(* Logix 5000 project; controller fun_probably 1769-L16ER-BB1B rev 34.12; software revision 34.01 *)

TASK MainTask (continuous, watchdog 500 ms) : MainProgram

MODULES
   Local : 1769-L16ER-BB1B (PointIO 0, rev 34.12)
      Discrete_IO : Embedded (PointIO 1, rev 34.11, Output RPI 20 ms)
END_MODULES

VAR_GLOBAL   (* controller tags *)
   ball_move : BOOL;
   ballSpeed : DINT;
   ballSpeedX : DINT := 4;
   ballSpeedY : DINT := 3;
   ballXpos : COUNTER := (ACC := 225);
   ballYpos : COUNTER := (ACC := 100);
   difficulty : TIMER := (PRE := 5000, ACC := 4915, EN := 1, TT := 1);
   direction : DINT;
   directionX : DINT := 1;
   directionY : DINT := 1;
   dX : DINT := 6;
   dY : DINT := -5;
   HMI_START : BOOL;
   ons1 : BOOL;
   ons2 : BOOL;
   ons3 : BOOL;
   ons4 : BOOL;
   ons5 : BOOL;
   refresh_rate : TIMER := (PRE := 50, ACC := 6, EN := 1, TT := 1);
   stop_start : COUNTER := (DN := 1);
   Xpos : DINT := 15;
   Xpos15 : DINT := 30;
   Xpos2 : DINT := 450;
   Xpos2_15 : DINT := 425;
   Xpos50 : DINT;
   Ypos : COUNTER := (ACC := 100);
   Ypos2 : COUNTER := (ACC := 100);
   Ypos2_50 : DINT := 150;
   Ypos50 : DINT := 150;
END_VAR

PROGRAM MainProgram   (* main routine MainRoutine *)

ROUTINE MainRoutine   (* ladder *)
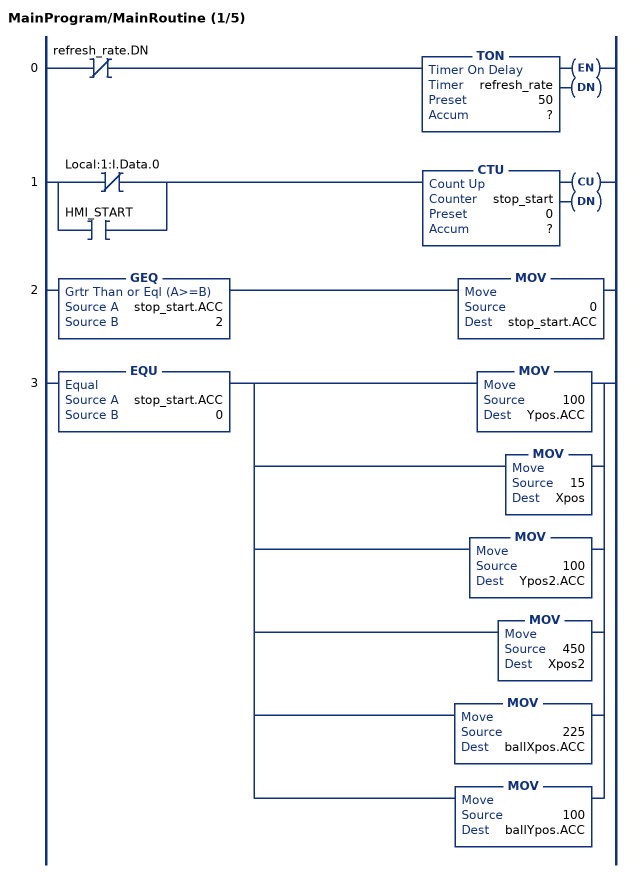
   0: XIO(refresh_rate.DN)TON(refresh_rate,?,?);
   1: [XIO(Local:1:I.Data.0) ,XIC(HMI_START) ]CTU(stop_start,?,?);
   2: GEQ(stop_start.ACC,2)MOV(0,stop_start.ACC);
   3: EQU(stop_start.ACC,0)[[MOV(100,Ypos.ACC) ,MOV(15,Xpos) ] ,[[MOV(100,Ypos2.ACC) ,MOV(450,Xpos2) ] ,[MOV(225,ballXpos.ACC) ,MOV(100,ballYpos.ACC) ] ] ];
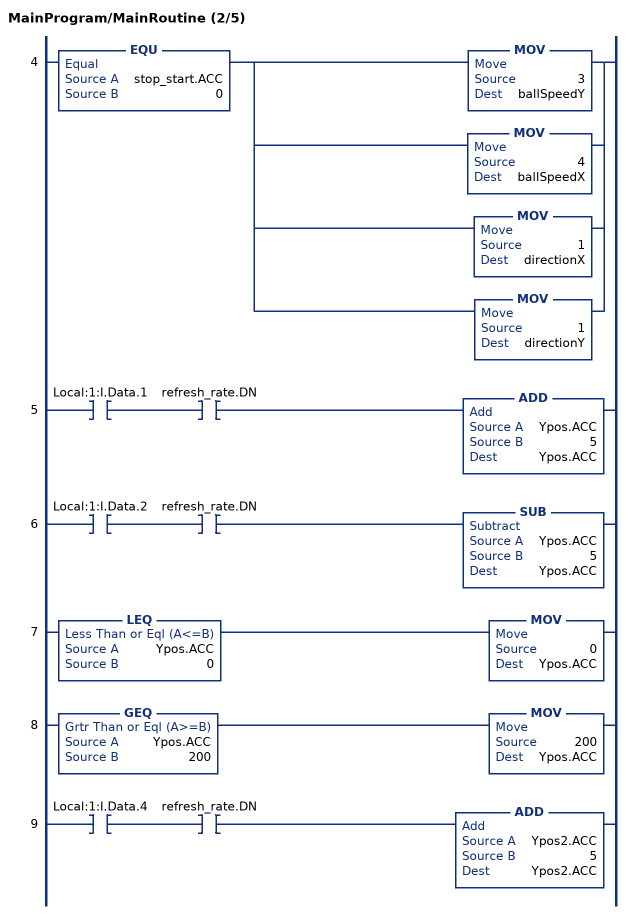
   4: EQU(stop_start.ACC,0)[MOV(3,ballSpeedY) ,[MOV(4,ballSpeedX) ,[MOV(1,directionX) ,MOV(1,directionY) ] ] ];
   5: XIC(Local:1:I.Data.1)XIC(refresh_rate.DN)ADD(Ypos.ACC,5,Ypos.ACC);
   6: XIC(Local:1:I.Data.2)XIC(refresh_rate.DN)SUB(Ypos.ACC,5,Ypos.ACC);
   7: LEQ(Ypos.ACC,0)MOV(0,Ypos.ACC);
   8: GEQ(Ypos.ACC,200)MOV(200,Ypos.ACC);
   9: XIC(Local:1:I.Data.4)XIC(refresh_rate.DN)ADD(Ypos2.ACC,5,Ypos2.ACC);
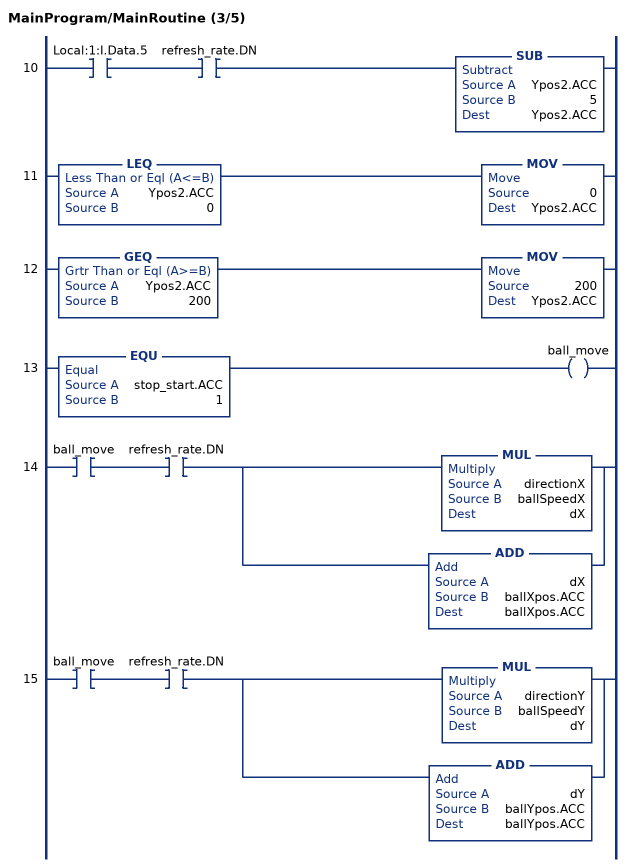
   10: XIC(Local:1:I.Data.5)XIC(refresh_rate.DN)SUB(Ypos2.ACC,5,Ypos2.ACC);
   11: LEQ(Ypos2.ACC,0)MOV(0,Ypos2.ACC);
   12: GEQ(Ypos2.ACC,200)MOV(200,Ypos2.ACC);
   13: EQU(stop_start.ACC,1)OTE(ball_move);
   14: XIC(ball_move)XIC(refresh_rate.DN)[MUL(directionX,ballSpeedX,dX) ,ADD(dX,ballXpos.ACC,ballXpos.ACC) ];
   15: XIC(ball_move)XIC(refresh_rate.DN)[MUL(directionY,ballSpeedY,dY) ,ADD(dY,ballYpos.ACC,ballYpos.ACC) ];
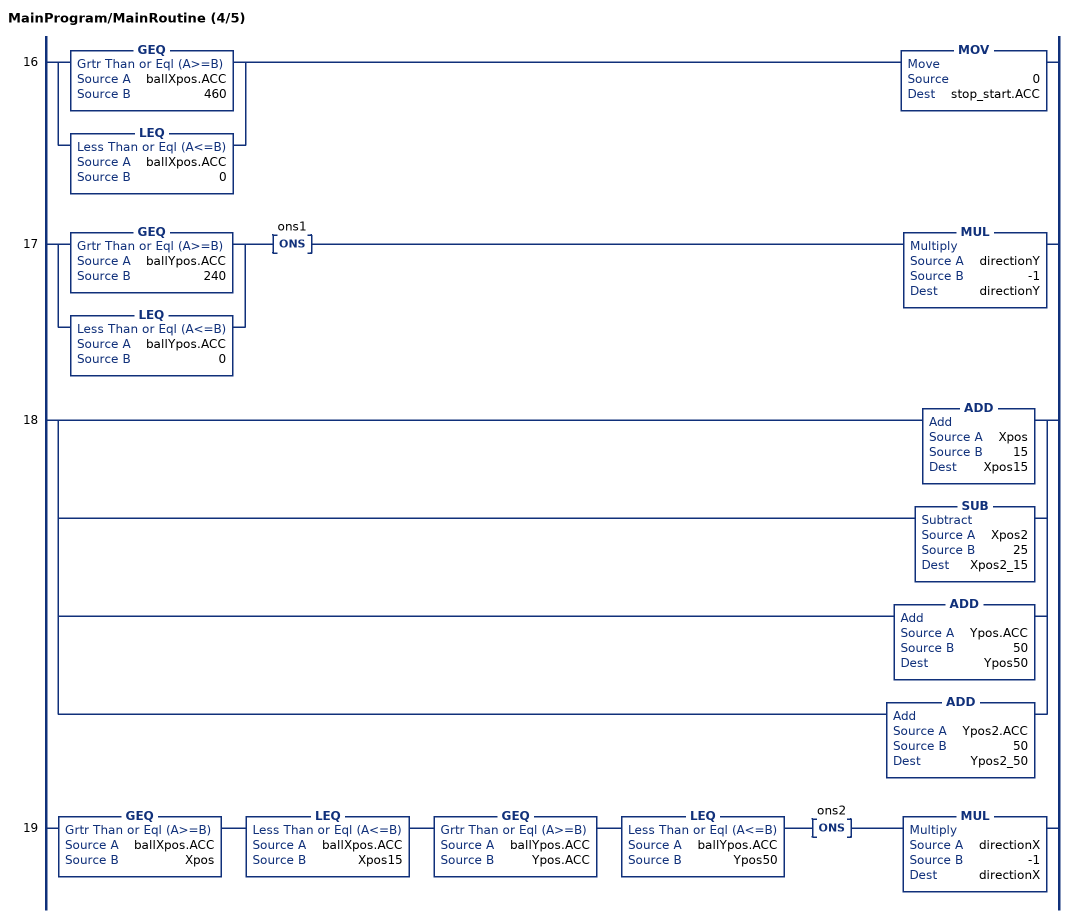
   16: [GEQ(ballXpos.ACC,460) ,LEQ(ballXpos.ACC,0) ]MOV(0,stop_start.ACC);
   17: [GEQ(ballYpos.ACC,240) ,LEQ(ballYpos.ACC,0) ]ONS(ons1)MUL(directionY,-1,directionY);
   18: [[ADD(Xpos,15,Xpos15) ,SUB(Xpos2,25,Xpos2_15) ] ,[ADD(Ypos.ACC,50,Ypos50) ,ADD(Ypos2.ACC,50,Ypos2_50) ] ];
   19: GEQ(ballXpos.ACC,Xpos)LEQ(ballXpos.ACC,Xpos15)GEQ(ballYpos.ACC,Ypos.ACC)LEQ(ballYpos.ACC,Ypos50)ONS(ons2)MUL(directionX,-1,directionX);
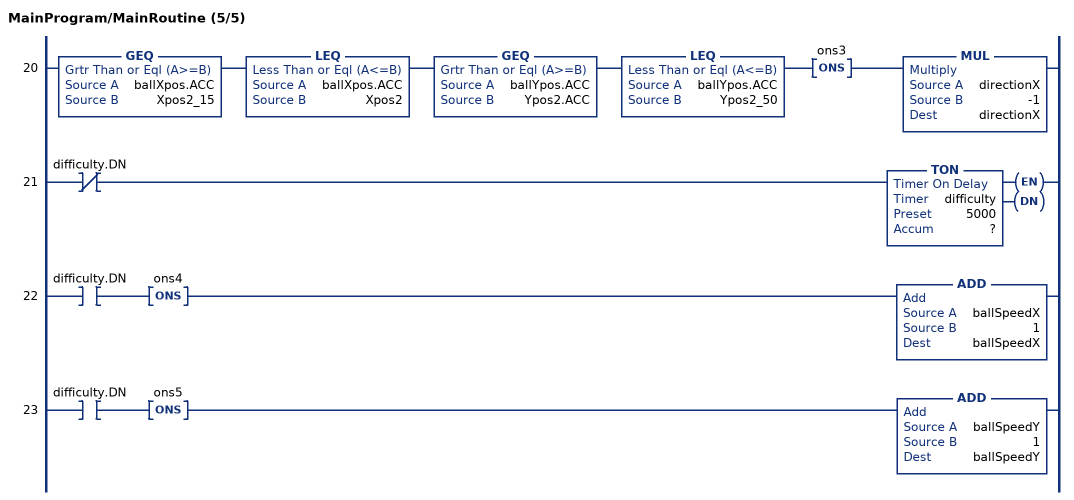
   20: GEQ(ballXpos.ACC,Xpos2_15)LEQ(ballXpos.ACC,Xpos2)GEQ(ballYpos.ACC,Ypos2.ACC)LEQ(ballYpos.ACC,Ypos2_50)ONS(ons3)MUL(directionX,-1,directionX);
   21: XIO(difficulty.DN)TON(difficulty,?,?);
   22: XIC(difficulty.DN)ONS(ons4)ADD(ballSpeedX,1,ballSpeedX);
   23: XIC(difficulty.DN)ONS(ons5)ADD(ballSpeedY,1,ballSpeedY);
END_ROUTINE

ROUTINE Test   (* structured text *)
   
END_ROUTINE
END_PROGRAM
